PROGRAM MAIN
VAR
	//Integrator
	ssMethodType : SINT := 1; 
	Timer : LREAL;
	
	//Pressure pA
	fbPressureGradient_pA : PressureGradient;
	PressurepA : LREAL;
	
	//Pressure pB
	fbPressureGradient_pB : PressureGradient;
	PressurepB : LREAL;
	
	//Pump
	fbPump : Pump;
	PumpTorque : LREAL;
	PumpFlowRate : LREAL;

	//OrificeEquation
	fbOrificeEquationQA : OrificeEquation;
	fbOrificeEquationQB : OrificeEquation;	
	OrificeFlow: LREAL;
	
	//HydraulicCylinder
	fbHydraulicCylinder : HydraulicCylinder;
	PressureBoreSide: LREAL;
	PressureRodSide: LREAL;
	AreaBoreSide: LREAL;
	AreaRodSide: LREAL;
	LoadForcePistonFL: LREAL;
	FrictionForce: LREAL;
	PistonMass: LREAL;

	
	pA : LREAL;
	pB : LREAL;
	qA : LREAL;
	qB : LREAL;
	ABore : LREAL;
	ARod : LREAL;
	xPos : LREAL;
	
END_VAR

//Timer
Timer := Timer + 0.01;

//Area Cylinder
ABore := EXPT(Param.DBore,2) * (Param.pi/4.0);
ARod := (EXPT(Param.DBore,2) - EXPT(Param.DRod,2)) * (Param.pi/4.0);

//Pressure Gradient pA and Pressure pA
fbPressureGradient_pA(
	TotalVolume := 2.9444E-04,
	BulkModulus := 10000.0,
	FlowrateIn := 60.0,
	FlowrateOut := 20.0,
	PressurePascal => PressurepA		//Pressure
	);
	
//Pressure Gradient pB and Pressure pB
fbPressureGradient_pB(
	TotalVolume := 2.9444E-04,
	BulkModulus := 10000.0,
	FlowrateIn := 60.0,
	FlowrateOut := 20.0,
	PressurePascal => PressurepB		//Pressure
	);

//Pump
fbPump(
	MotorSpeedRPM := 413.2,
	PumpDisplacement := 10.6E-6,
	DeltaMaxPressure := 250.0,
	PumpTorque => PumpTorque,
	PumpFlowRate => PumpFlowRate
	);
	
//OrificeEquationA (Q_A)
fbOrificeEquationQA(
	PressureOut := pA, 			//Found value from old simulink project, this one goes to the tank i guess
	PressureIn := 180,		
	Kv := 1,
	ValveOpening := 1,	
	OrificeFlow => OrificeFlow
	);
	
//OrificeEquationB (Q_B)
fbOrificeEquationQB(
	PressureOut := pB, 			//Found value from old simulink project, this one goes to the tank i guess
	PressureIn := 180,		
	Kv := 1,
	ValveOpening := 1,
	OrificeFlow => OrificeFlow
	);

END_PROGRAM

(* stored: Version 1.1.0.1, ProductVersion 3.1.4024.9
   POU MAIN: Id {d1c7ef4e-0337-49c7-9736-af80a39f1b25}, SpecialFunc None *)
